// Mitsubishi GX Works2 project: slave   PLC: FX3U/FX3UC

PROGRAM MAIN
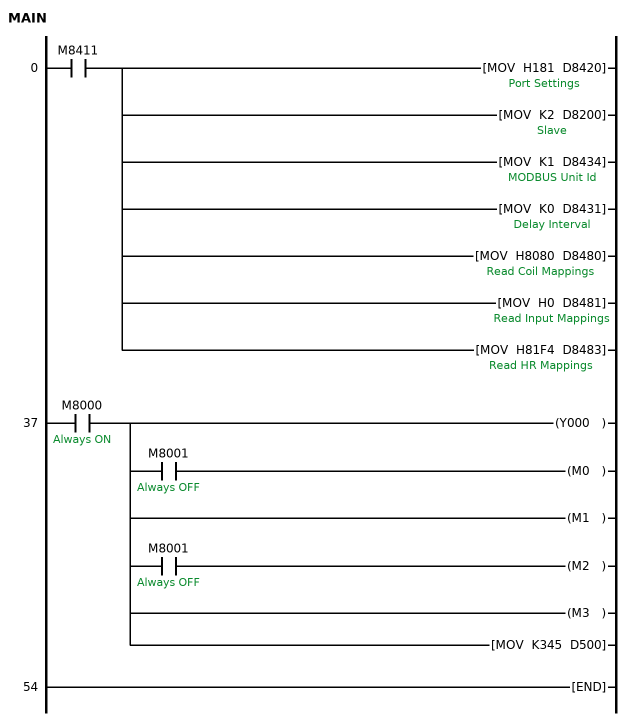
0     LD      M8411
      MOV     H181 D8420  ; Port Settings
      MOV     K2 D8200  ; Slave
      MOV     K1 D8434  ; MODBUS Unit Id
      MOV     K0 D8431  ; Delay Interval
      MOV     H8080 D8480  ; Read Coil Mappings
      MOV     H0 D8481  ; Read Input Mappings
      MOV     H81F4 D8483  ; Read HR Mappings
37    LD      M8000  ; Always ON
      OUT     Y000
      MPS
      AND     M8001  ; Always OFF
      OUT     M0
      MPP
      OUT     M1
      MPS
      AND     M8001  ; Always OFF
      OUT     M2
      MPP
      OUT     M3
      MOV     K345 D500
54    END
END_PROGRAM
